// Mitsubishi GX Works2 project: 240528_사칙연산1   PLC: Q03UDV

PROGRAM MAIN
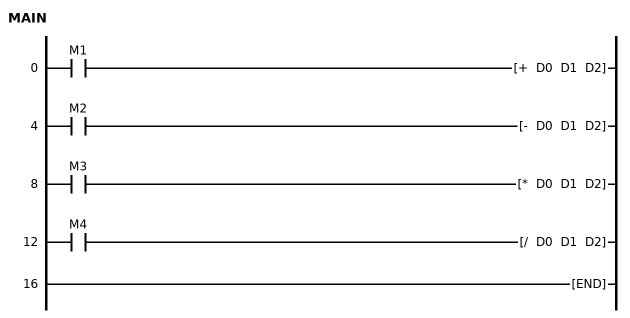
0     LD      M1
      +       D0 D1 D2
4     LD      M2
      -       D0 D1 D2
8     LD      M3
      *       D0 D1 D2
12    LD      M4
      /       D0 D1 D2
16    END
END_PROGRAM
